(* IEC 61131-3 sources: rules_plc/examples/interface_deps, 3 files *)

(* ---- plant.st ---- *)
(* Production code -- calls Pump from vendor_pump.st via
interface_deps, so vendor_pump.st is visible to plc's `-i` at
compile time (for cross-library type resolution) but does NOT ride
along in the exported StInfo.compilation_context.sources bucket
(see examples/interface_deps/remote_manifest.bzl). *)

FUNCTION_BLOCK Plant
    VAR_INPUT
        rIn : REAL;
    END_VAR
    VAR_OUTPUT
        rOut : REAL;
    END_VAR
    VAR
        pump : Pump;
    END_VAR
    pump(rIn := rIn);
    rOut := pump.rOut;
END_FUNCTION_BLOCK

(* ---- vendor_pump.st ---- *)
(* Vendor-supplied interface. In production this file would ship from
an upstream vendor Bazel module carrying only {external}
declarations of the POUs the vendor's runtime provides -- never
their bodies. plc emits an extern declaration for the FB (plus its
struct layout in the generated headers) and skips code generation
for its body.

    The body is supplied here by vendor_pump_stub.cc through cc_deps,
    for local exercise under the locally-installed plc without any
        real vendor runtime.

        In the source-bucket model, this st_library IS "vendor territory":
        consumers pull it in through `interface_deps`, so its
        `vendor_pump.st` sits in StInfo.compilation_context.interface_sources
    (visible to plc's `-i` at compile time for cross-library type
        resolution, never uploaded to the remote plc, which already has the
        vendor's real impl). *)

        {external}
        FUNCTION_BLOCK Pump
            VAR_INPUT
                rIn : REAL;
            END_VAR
            VAR_OUTPUT
                rOut : REAL;
            END_VAR
        END_FUNCTION_BLOCK

(* ---- main_program.st ---- *)
PROGRAM main_program
    VAR
        plant : Plant;
    END_VAR

    plant(rIn := 21.0);
END_PROGRAM
